FUNCTION_BLOCK FB_DRIFTCONTROL
VAR_INPUT
  bI_Reset                    : BOOL;            (*reset fb and controller*)
  bI_ReceiptMessage           : BOOL;            (*reset error*)
  bI_Enable                   : BOOL;            (*[internal] auto enable of control*)
  bI_OutputEnable             : BOOL;            (*enable control output or 1.0 if off*)
  bI_RegisterMark             : BOOL;            (*start trigger (e.g. register mark)*)
  
  lI_RegisterMarkPosition     : DINT;            (*[Subpixel] Mark position*)
  lI_RefPosition              : DINT;            (*[Subpixel] Refereence position*)
  lI_ImgPosition              : DINT;            (*[Subpixel] Image position*)
(*UNUSED*)  fI_RefPosition            : LREAL;          (*[um] Refereence position*)    
(*UNUSED*)  fI_ImgPosition            : LREAL;          (*[um] Image position*)

  iI_Res_Ph                   : INT;             (*[dpi] resolution printhead native*)
  iI_Res_SubPix               : INT;             (*[-] resolution subpixel*)
  pI_JobSettings              : POINTER TO ST_JobSettings;
  
  fI_TaskCycleTime            : REAL;            (*Task cycle time of actual task [s]*)
END_VAR

VAR_OUTPUT
  fO_SpeedCorrectionFactor    : LREAL;           (*[-] controller output*)
  bO_ContrErr                 : BOOL;            (*correction fail (out of bound)*)
  bO_SupervisionContrErr      : BOOL;            (*supervision (out of bound)*)
  bO_SupervisionMissMarks     : BOOL;            (*supervision misses marks after X cycles*)
  bO_ControllerAdjusted       : BOOL;            (*controller adjusted after X cycles*)
END_VAR

VAR
  bL_ControlActive            : BOOL;
  nL_CountCyclesToAdjust      : INT;             (*Count number of cycles to adjust the controller*)
  bL_RegisterMark             : BOOL;
  
  lL_LastRegisterMarkPosition : DINT;            (*[SubPixel] last stored mark position*)
  lL_LastRefPosition          : DINT;            (*[Subpixel] Refereence position*)
  lL_LastImgPosition          : DINT;            (*[Subpixel] Image position*)

  fL_RefSpeed                 : LREAL;           (*[rev/s] : rev ^= image, revolution of reference axe sync with image*)
  fL_ImgSpeed                 : LREAL;           (*[rev/s] : rev ^= image, revolution of reference axe sync with image*)
  fL_RefLength                : LREAL;           (*[Subpixel in float!] real length of one image = reference distance between print marks*)
  fL_RefLengthMM              : LREAL;           (*[mm] real length of one image = reference distance between print marks*)
  lL_ImgLength                : DINT;            (*[Subpixel] image length of job*)
  fL_RefPos                   : LREAL;           (*[rev] : 1rev ^= 1ImageLength, number rev after start*)
  fL_ImgPos                   : LREAL;           (*[rev] : 1rev ^= 1ImageLength, number rev after start*)
  fL_LastRefPos               : LREAL;           (*[rev] : 1rev ^= 1ImageLength, number rev after start*)
  fL_LastImgPos               : LREAL;           (*[rev] : 1rev ^= 1ImageLength, number rev after start*)
  fL_ShiftPos                 : LREAL;           (*[rev] shift position rev->img*)

  fL_DeltaCtrl                : LREAL;           (**)
  fL_CtrlGainFactor           : LREAL;           (**)
        
  fL_DeltaTimeStamp           : LREAL;           (**)
  tL_CurrentTimeStamp         : T_DCTIME64;      (* Get Current Timestamp *)
  tL_LastTimeStamp            : T_DCTIME64;      (* Get Current Timestamp *)
  fB_PID                      : FB_BasicPID;     (**)
  iL_State                    : UINT;            (**)

  bL_FormatWarning            : BOOL;
  bL_Error                    : BOOL;
  bL_RegisterEvent            : BOOL;
  bL_ResetInternal            : BOOL;            (*internal reset*)
  fL_DeltaLength              : LREAL;           (*image length difference between img and ref bewtween a cycle*)
  lL_ConversionErrorCtr       : UDINT;

  bL_SupervisionContrErr      : BOOL;            (*supervision (out of bound)*)
  fb_TonSupervisionContrErr   : TON;             (*supervision (out of bound)*)
  fb_TonSupervisionMarkErr    : TON;             (*supervision marks missing*)
  fb_TonSupervisionMissMarkErr: TON;             (*supervision marks missing*)

  fC_MaxCorrection            : LREAL := 1.10;  (*moved from Constant: org value: 1.05*)
  fC_MinCorrection            : LREAL := 0.90;  (*moved from Constant: org value: 0.95*)
  fC_MaxControlError          : LREAL := 0.2;   (*moved from Constant: org value: 0.1*)
END_VAR

VAR CONSTANT
  fC_NormSpeedCorrectionFactor: LREAL := 1.0;
  
  fC_MaxFormatDifference      : LREAL := 1.0;
  
  fC_MaxFormatLength          : LREAL := 1.0;       (*m*)
  fC_MinSubstrateSpeed        : LREAL := 5.0/60.0 ; (*m/s*)
  lC_MaxFormatLength          : DINT  := LREAL_TO_DINT(fC_MaxFormatLength/0.0254*32*600);  (*Subpixel*)
  fC_MaxCycleTime             : LREAL := fC_MaxFormatLength/fC_MinSubstrateSpeed;  (*sec*)
END_VAR

VAR PERSISTENT
  fR_SpeedCorrectionWindow    : LREAL := 0.05;     (*Supervision window*)
  tR_SpeedCorrectionTime      : TIME  := T#10S;    (*Supervision time*)

  fI_ControllerPGain          : LREAL := 0.5;      (*PDI controller P-Gain*)
  fI_ControllerIGain          : LREAL := 20;       (*PDI controller I-Gain*)
  fI_DriftTimeShift           : LREAL;             (*[ms] register shift time*)
  nI_NbCyclesToAdjust         : INT   := 0;        (*Number of cycles to adjust the controller*)
  nI_NbMissMarksToStop        : INT   := 5;        (*Number of missed marks to stop the machine*)
END_VAR

(*--- Reset*)
IF bI_Reset OR bL_ResetInternal THEN
  iL_State := 0;
END_IF;

(*--- Reset error*)
IF bI_ReceiptMessage THEN
  bO_SupervisionMissMarks := FALSE;
END_IF;

(*--- cyclic called on register event*)
IF bI_RegisterMark AND NOT bL_RegisterMark THEN
  bL_RegisterEvent    := TRUE;
  tL_CurrentTimeStamp := F_GetCurDcTaskTime64();
  fL_DeltaTimeStamp   := (ULINT_TO_LREAL(tL_CurrentTimeStamp) - ULINT_TO_LREAL(tL_LastTimeStamp)) * 0.000_000_001;
ELSE
  bL_RegisterEvent    := FALSE;
END_IF


// ----- State machine 
CASE iL_State OF
  000:  (*Reset --------------------*)
    bL_ControlActive := FALSE;
    fB_PID(bReset := TRUE);
    fO_SpeedCorrectionFactor := 1.0; 
    fB_PID.bReset := FALSE;
    fL_RefPos := 0;
    fL_ImgPos := 0;
    bL_SupervisionContrErr := FALSE;
    bO_SupervisionContrErr := FALSE;
    bO_SupervisionMissMarks:= FALSE;

    IF pI_JobSettings <> 0 THEN
      iL_State:=001;
    ELSE
      iL_State:=000;
    END_IF

    nL_CountCyclesToAdjust := 0;
    bO_ControllerAdjusted  := (nI_NbCyclesToAdjust = 0);
    bL_ControlActive       := FALSE;
    bL_Error               := FALSE;
    bI_Enable              := FALSE; (*Disable by default*)
    bO_ContrErr            := FALSE;

    (*Check for missing marks*)
    fb_TonSupervisionMissMarkErr(IN := FALSE);
    
  001:  (*Control Disabled --------------------*)
    (*New PrintLib 1.5.2.6
    lL_ImgLength:=UDINT_TO_DINT(pI_JobSettings^.lI_ImageDepth)*iI_Res_SubPix; *)
    lL_ImgLength := FC_CONV_M_TO_SUBPX( UDINT_TO_LREAL(pI_JobSettings^.lI_ImageDepth) / 1_000_000
                                      , iI_Res_Ph
                                      , iI_Res_SubPix);

    IF pI_JobSettings^.lI_PrintMode.ePr_PRINT_MODE_ENDLESS THEN
      bI_Enable:=TRUE; (*Automatically enable in Endless Mode*)
    END_IF    
    
    IF bI_Enable AND (fL_DeltaTimeStamp < fC_MaxCycleTime) AND bL_RegisterEvent AND lL_ImgLength >0 THEN (*Enabled and moving*)
      iL_State:=010;
    ELSE
      (*Check for missing marks*)
      fb_TonSupervisionMissMarkErr(IN := bI_OutputEnable, PT := LREAL_TO_TIME(fL_DeltaTimeStamp * 1000 * nI_NbMissMarksToStop));
      IF fb_TonSupervisionMissMarkErr.Q THEN
        bO_SupervisionMissMarks := TRUE;

        iL_State:=099;
      ELSE 
        iL_State:=001;
      END_IF
    END_IF

    fO_SpeedCorrectionFactor := 1.0; 
    nL_CountCyclesToAdjust   := 0;
    bO_ControllerAdjusted    := (nI_NbCyclesToAdjust = 0);

  010:  (*Starting Controller ------------------*)
    IF (fL_DeltaTimeStamp > fC_MaxCycleTime) THEN
      iL_State:=001;
    ELSIF bL_RegisterEvent THEN
      (*registered first label*)
      fL_RefLength := DINT_TO_LREAL(lI_RegisterMarkPosition - lL_LastRegisterMarkPosition);
      (*New PrintLib 1.5.2.6
      lL_ImgLength:=UDINT_TO_DINT(pI_JobSettings^.lI_ImageDepth)*iI_Res_SubPix; *)
      lL_ImgLength := FC_CONV_M_TO_SUBPX( UDINT_TO_LREAL(pI_JobSettings^.lI_ImageDepth) / 1_000_000
                                        , iI_Res_Ph
                                        , iI_Res_SubPix);
      
      IF fL_RefLength > 0 AND lL_ImgLength > 0 THEN
        IF DINT_TO_LREAL(ABS(FC_LREAL_TO_DINT(fL_RefLength)-lL_ImgLength)*100)/fL_RefLength > fC_MaxFormatDifference THEN
          bL_FormatWarning:=TRUE;
        ELSE
          bL_FormatWarning:=FALSE;
        END_IF
        iL_State  := 020;
        fL_RefPos := 0;
        fL_ImgPos := 0;
        (*Check for missing marks*)
        fb_TonSupervisionMarkErr    (IN := FALSE);
        fb_TonSupervisionMissMarkErr(IN := FALSE);
      ELSE
        iL_State:=099;
      END_IF
    ELSE
      iL_State:=010;
    END_IF
    
    fL_CtrlGainFactor := 1.0;
    bL_ControlActive  := FALSE;
    
  020:  (*Controller enabled--------------------*)
    
    IF bL_RegisterEvent THEN (*run controller when a mark trigger was detected*)
      (*Check for missing marks*)
      fb_TonSupervisionMarkErr    (IN := FALSE);
      fb_TonSupervisionMissMarkErr(IN := FALSE);
    
      (*Wait until controller is stable*)
      IF (nL_CountCyclesToAdjust < nI_NbCyclesToAdjust) THEN
        nL_CountCyclesToAdjust := nL_CountCyclesToAdjust + 1;
      END_IF

      (*position in [rev] from beginning*)
      fL_RefLength := DINT_TO_LREAL(lI_RegisterMarkPosition - lL_LastRegisterMarkPosition);
      IF fL_RefLength > 0 THEN
        fL_RefPos := fL_LastRefPos + DINT_TO_LREAL(lI_RefPosition - lL_LastRefPosition) / fL_RefLength;
        fL_ImgPos := fL_LastImgPos + DINT_TO_LREAL(lI_ImgPosition - lL_LastImgPosition) / DINT_TO_LREAL(lL_ImgLength);  
      END_IF

      (*calculate current speed of ref and img position*)
      (*    'traveled pos in cycle' / ('Reference Length sampled' / 'time diff sampled' *)
      fL_RefSpeed := (fL_RefPos - fL_LastRefPos) / fL_DeltaTimeStamp;
      fL_ImgSpeed := (fL_ImgPos - fL_LastImgPos) / fL_DeltaTimeStamp;   
    
//      fL_RefSpeed:=DINT_TO_LREAL(lI_RefPosition-lL_LastRefPosition)/(fL_RefLength*fL_DeltaTimeStamp);
//      fL_ImgSpeed:=DINT_TO_LREAL(lI_ImgPosition-lL_LastImgPosition)/(DINT_TO_LREAL(lL_ImgLength)*fL_DeltaTimeStamp);    
//      fL_RefPos:=0.000001*fI_RefPosition/( fL_RefLength / INT_TO_REAL(iI_Res_Ph * iI_Res_SubPix) * 0.0254);
//      fL_ImgPos:=0.000001*fI_ImgPosition/FC_CONV_SUBPX_TO_M(lL_ImgLength,INT_TO_UDINT(iI_Res_Ph),INT_TO_UDINT(iI_Res_SubPix));
      
      (*shift calculation*)
      fL_ShiftPos := (fI_DriftTimeShift / 1000) * fL_RefSpeed;
      
      (*calc control diff*)
      fL_DeltaCtrl := (fL_RefPos - fL_ImgPos) + fL_ShiftPos;
      
      (*controller*)
      fB_PID.fCtrlCycleTime  := fL_DeltaTimeStamp;  // use fI_TaskCycleTime if running controller cyclically
      fB_PID.bReset          := FALSE;
      fB_PID.fSetpointValue  := fL_DeltaCtrl;
      fB_PID.fActualValue    := 0.0;
      fB_PID.fKp             := fI_ControllerPGain * fL_CtrlGainFactor;
      fB_PID.fTd             := 0.0;
      fB_PID.fTn             := fI_ControllerIGain;
      fB_PID.fTv             := 0.0;

      fB_PID();
    END_IF
    
    IF bI_OutputEnable THEN
      fO_SpeedCorrectionFactor := fB_PID.fCtrlOutput + 1.0;
    ELSE
      fO_SpeedCorrectionFactor := 1.0;
    END_IF;

    IF fO_SpeedCorrectionFactor > fC_MaxCorrection THEN
      fO_SpeedCorrectionFactor := fC_MaxCorrection;
      fL_CtrlGainFactor := 0.1;  (*TODO ARW*)
      bO_ContrErr       := TRUE;
    ELSIF fO_SpeedCorrectionFactor < fC_MinCorrection THEN
      fO_SpeedCorrectionFactor := fC_MinCorrection;
      fL_CtrlGainFactor := 0.1;  (*TODO ARW*)
      bO_ContrErr       := TRUE;
    ELSE
      fO_SpeedCorrectionFactor := fO_SpeedCorrectionFactor;
      fL_CtrlGainFactor := 1;
      bO_ContrErr       := FALSE;
    END_IF
    (*Supervision*)
    IF fO_SpeedCorrectionFactor > (fC_NormSpeedCorrectionFactor + fR_SpeedCorrectionWindow) THEN
      bL_SupervisionContrErr := TRUE;
    ELSIF fO_SpeedCorrectionFactor < (fC_NormSpeedCorrectionFactor - fR_SpeedCorrectionWindow) THEN
      bL_SupervisionContrErr := TRUE;
    ELSE
      bL_SupervisionContrErr := FALSE;
    END_IF
    fb_TonSupervisionContrErr( IN := bL_SupervisionContrErr, PT := tR_SpeedCorrectionTime);
    bO_SupervisionContrErr := fb_TonSupervisionContrErr.Q;

    (*Check for missing marks*)
    fb_TonSupervisionMarkErr    (IN := TRUE, PT := LREAL_TO_TIME(fL_DeltaTimeStamp * 1000 * 2)); (*[s] to [ms] and factor of 2*)
    fb_TonSupervisionMissMarkErr(IN := TRUE, PT := LREAL_TO_TIME(fL_DeltaTimeStamp * 1000 * nI_NbMissMarksToStop)); (*[s] to [ms] and factor of the setting*)
    
    (*Check for errors  while control was on*)
    IF ((fL_DeltaTimeStamp > fC_MaxCycleTime) OR (fL_DeltaCtrl > fC_MaxControlError) OR fL_RefLength=0) AND bL_RegisterEvent THEN
      iL_State:=099;
    ELSIF NOT bI_Enable OR fb_TonSupervisionMarkErr.Q THEN
      iL_State:=030;  
    ELSE
      iL_State:=020;
    END_IF

    bL_ControlActive      := TRUE;
    bO_ControllerAdjusted := (nL_CountCyclesToAdjust >= nI_NbCyclesToAdjust) OR (nI_NbCyclesToAdjust = 0);

  030:  (*Stopping controller-------------------*)
    iL_State                 := 001;  
    bL_ControlActive         := FALSE;
    fO_SpeedCorrectionFactor := 1.0;
    bO_ContrErr              := FALSE;
    
  099:  (*Error---------------------------------*)
    bL_Error                 := TRUE;
    bL_ControlActive         := FALSE;
    fO_SpeedCorrectionFactor := 1.0; 
    bO_ContrErr              := FALSE;
END_CASE

fL_RefLengthMM := FC_CONV_SUBPX_TO_M( LREAL_TO_DINT(fL_RefLength), INT_TO_UDINT(iI_Res_Ph), INT_TO_UDINT(iI_Res_SubPix)) * 1_000;

(*--- cyclic called on register event*)
IF bL_RegisterEvent OR bI_Reset THEN
  (*save old values & debug*)
  fL_DeltaLength              := lL_ImgLength - fL_RefLength;  (*debug only*)
  lL_LastRegisterMarkPosition := lI_RegisterMarkPosition; 
  lL_LastRefPosition          := lI_RefPosition;       (*used for speed only*)
  lL_LastImgPosition          := lI_ImgPosition;       (*used for speed only*)
  tL_LastTimeStamp            := tL_CurrentTimeStamp;
  fL_LastRefPos               := fL_RefPos;
  fL_LastImgPos               := fL_ImgPos;
END_IF;

END_FUNCTION_BLOCK

(* stored: Version 1.1.0.1, ProductVersion 3.1.4024.11
   POU FB_DRIFTCONTROL: Id {525b6909-7917-44ad-af97-c164fbbd270b}, SpecialFunc None *)
